KUKA KRL program: C3_GHvH.src, C3_GHvH.dat

--- C3_GHvH.src ---
2&ACCESS RV1
DEF  C3_GHvH (GR:IN, WP:IN)
   ; GR [GRAVITY], WP [WHO PLAYS], FG [FIELD GAME]
   ; FP1 [FIELD PLAYER 1], FP2 [FIELD PLAYER 2]

   ; ### DECLARATION ###
   DECL INT GR, WP
   DECL FRAME FG[4, 6]
   DECL FRAME FPL1[2, 6], FPL2[2, 6]

   STRUC CUBE INT player, INT pos_x, INT pos_y, INT round
   DECL CUBE FIELD[4, 6]

   DECL BOOL playing, victory
   DECL INT gameround, temp
   DECL INT row, col

   DECL INT sel_row, sel_col

   DECL REAL Player1X, Player1Y, Player1Z
   DECL REAL Player2X, Player2Y, Player2Z
   DECL REAL FX, FY, FZ

   DECL FRAME START_POS_P1, START_POS_P2  ; ABLAGE Player 1, Player 2
   DECL FRAME START_POS_FIELD             ; Spielfeld

   DECL INT j, i

   ;FOLD INI;%{PE}
      ;FOLD BASISTECH INI
         GLOBAL INTERRUPT DECL 3 WHEN $STOPMESS==TRUE DO IR_STOPM ( )
         INTERRUPT ON 3
         BAS (#INITMOV,0 )
      ;ENDFOLD (BASISTECH INI)
      ;FOLD USER INI
         ;Make your modifications here

      ;ENDFOLD (USER INI)
   ;ENDFOLD (INI)

   ;FOLD PTP HOME  Vel= 100 % DEFAULT;%{PE}%MKUKATPBASIS,%CMOVE,%VPTP,%P 1:PTP, 2:HOME, 3:, 5:100, 7:DEFAULT
      $BWDSTART = FALSE
      PDAT_ACT=PDEFAULT
      FDAT_ACT=FHOME
      BAS (#PTP_PARAMS,100 )
      $H_POS=XHOME
      PTP  XHOME
   ;ENDFOLD


   ; ### INIT ###
   playing = TRUE
   gameround = 1


   ; ### FIELD FILLING ###
   Player1X = 82.2353058
   Player1Y = -41.7172813
   Player1Z = 0.388017595

   Player2X = 83.7938
   Player2Y = 161.979172
   Player2Z = -2.58887553

   START_POS_P1 = XP1
   START_POS_P2 = XP2

   FOR j = 0 TO 1 STEP 1
       FOR i = 0 TO 5 STEP 1
          $BASE = base_data[6]
          $TOOL = tool_data[14]

          START_POS_P1.X = Player1X - j*46.8868446
          START_POS_P1.Y = Player1Y + i*31.2624015

          START_POS_P2.X = Player2X - j*46.8868446
          START_POS_P2.Y = Player2Y + i*31.2624015

          FPL1[j + 1, i + 1] = START_POS_P1
          FPL2[j + 1, i + 1] = START_POS_P2

       ENDFOR
    ENDFOR

    FX = 199.0000
    FY = 3.00000
    FZ = -0.367093951

    START_POS_FIELD = XP3
    ; FIELD
    FOR j = 0 TO 3 STEP 1
       FOR i = 0 TO 5 STEP 1
          ; X = 31.410049
          ; y = 46.55986355

          START_POS_FIELD.X = FX - j*31.410049
          START_POS_FIELD.Y = FY + i*46.55986355

          FG[j +1, i + 1] = START_POS_FIELD

       ENDFOR
    ENDFOR


    ; ## FIELD ( Belegungsinformationen ) initial füllen
    FOR j = 0 TO 3
       FOR i = 0 TO 5
          FIELD[j+1, i+1].player = -1
          FIELD[j+1, i+1].pos_x = -1
          FIELD[j+1, i+1].pos_y = -1
          FIELD[j+1, i+1].round = -1
       ENDFOR
    ENDFOR

   ; ### GAMELOOP ###

   WHILE playing and (gameround <= 24) and ($IN[1] == False)

      ;-> hole Stein von Spieler WP
      ; Y POS
      row = 1
      col = gameround

      ; X POS
      IF gameround > 12 THEN
         row = 2
         col = gameround - 12
      ENDIF

      col = (col+1) / 2

      IF WP == 1 THEN
         $OUT[1] = TRUE
         C3_getcube(FPL1[row, col])
      ELSE
         $OUT[2] = TRUE
         C3_getcube(FPL2[row, col])
      ENDIF

      ;-> Auswahl auf Pad
      ; Test Gravity = off
      sel_row = 0
      while sel_row == 0

         sel_col = C3_IO(4)
         if GR == 1 then
            FOR j = 1 TO 4 STEP 1
               IF FIELD[j, sel_col].player == -1 THEN
                  sel_row = j
               ENDIF
            ENDFOR
         if sel_row == 0 then
             temp = C3_IO(8)
         endif
         ELSE
            sel_row = C3_IO(5)
            IF FIELD[sel_row, sel_col].player <> -1 THEN
               temp = C3_IO(8)
               sel_row = 0
            ENDIF
         ENDIF

      ENDWHILE


      ;-> Setze Stein
      C3_placecube(FG[sel_row, sel_col])

      ; Field[reihe, spalte] = Cube(whoPlays, reihe, spalte, gameround) - TODO
      FIELD[sel_row, sel_col].player = WP
      FIELD[sel_row, sel_col].pos_x = sel_row
      FIELD[sel_row, sel_col].pos_y = sel_col
      FIELD[sel_row, sel_col].round = gameround

      ;Prüfe ob Spieler gewonnen hat
      victory = C3_checkVictory(FIELD[,], WP)
      if victory then
         ; PLAYER X won
         gameround = C3_IO(WP + 5)
         playing = False
      ENDIF

      ;-> Prüfe Gewinn (Ja -> Anzeige und loop beenden, nein -> weiter)

      ; Player wechseln
      IF WP == 1 THEN
         $OUT[1] = FALSE
         $OUT[2] = TRUE
         WP = 2
      ELSE
         $OUT[2] = FALSE
         $OUT[1] = TRUE
         WP = 1
      ENDIF

      gameround = gameround + 1

   ENDWHILE

   ;-> Setze Steine zurück
   C3_cleanup(FIELD[,], FPL1[,], FPL2[,], FG[,])

   ;FOLD PTP HOME  Vel= 100 % DEFAULT;%{PE}%MKUKATPBASIS,%CMOVE,%VPTP,%P 1:PTP, 2:HOME, 3:, 5:100, 7:DEFAULT
      $BWDSTART = FALSE
      PDAT_ACT=PDEFAULT
      FDAT_ACT=FHOME
      BAS (#PTP_PARAMS,100 )
      $H_POS=XHOME
      PTP  XHOME
   ;ENDFOLD
END

--- C3_GHvH.dat ---
&ACCESS RV1
DEFDAT  C3_GHvH
;FOLD EXTERNAL DECLARATIONS;%{PE}%MKUKATPBASIS,%CEXT,%VCOMMON,%P
;FOLD BASISTECH EXT;%{PE}%MKUKATPBASIS,%CEXT,%VEXT,%P
EXT  BAS (BAS_COMMAND  :IN,REAL  :IN )
;ENDFOLD (BASISTECH EXT)
;FOLD USER EXT;%{E}%MKUKATPUSER,%CEXT,%VEXT,%P
;Make your modifications here

DECL E6POS XP1={X 82.2353058,Y -41.7172813,Z 0.388017595,A -27.1446362,B -89.7355,C 117.001740,S 2,T 34,E1 0.0,E2 0.0,E3 0.0,E4 0.0,E5 0.0,E6 0.0}
DECL FDAT FP1={TOOL_NO 14,BASE_NO 6,IPO_FRAME #BASE,POINT2[] " ",TQ_STATE FALSE}
DECL PDAT PPDAT1={VEL 100.000,ACC 100.000,APO_DIST 100.000,GEAR_JERK 50.0000,EXAX_IGN 0}

DECL E6POS XP2={X 83.7938,Y 161.979172,Z -2.58887553,A -27.3082161,B -89.7352,C 117.165596,S 2,T 35,E1 0.0,E2 0.0,E3 0.0,E4 0.0,E5 0.0,E6 0.0}
DECL FDAT FP2={TOOL_NO 14,BASE_NO 6,IPO_FRAME #BASE,POINT2[] " ",TQ_STATE FALSE}
DECL PDAT PPDAT2={VEL 100.000,ACC 100.000,APO_DIST 100.000,GEAR_JERK 50.0000,EXAX_IGN 0}

DECL E6POS XP3={X 197.537445,Y 1.61035585,Z -0.367093951,A -176.990829,B -88.1367340,C 176.297943,S 2,T 10,E1 0.0,E2 0.0,E3 0.0,E4 0.0,E5 0.0,E6 0.0}
DECL FDAT FP3={TOOL_NO 14,BASE_NO 6,IPO_FRAME #BASE,POINT2[] " ",TQ_STATE FALSE}
DECL PDAT PPDAT3={VEL 100.000,ACC 100.000,APO_DIST 100.000,GEAR_JERK 50.0000,EXAX_IGN 0}

;ENDFOLD (USER EXT)
;ENDFOLD (EXTERNAL DECLARATIONS)
ENDDAT
